{attribute 'linkalways'} 
{attribute 'no_explicit_call' := 'This FB is a CLASS and must be accessed using methods or properties'}
{attribute 'enable_dynamic_creation'}
FUNCTION_BLOCK FINAL NOT_ULINT EXTENDS Node
VAR
	in : _ULINT(0);
	out : _ULINT(0);
END_VAR

METHOD PUBLIC Clone : I_Node
VAR
	pNode : POINTER TO NOT_ULINT;
END_VAR
pNode := __NEW(NOT_ULINT);
Clone := pNode^;
END_METHOD

METHOD FB_init : BOOL
VAR_INPUT
	bInitRetains : BOOL; // if TRUE, the retain variables are initialized (warm start / cold start)
	bInCopyCode : BOOL;  // if TRUE, the instance afterwards gets moved into the copy code (online change)
END_VAR
AddInput('in',THIS^.in);
AddOutput('out', THIS^.out);
END_METHOD

METHOD PROTECTED OnExecute
VAR
END_VAR
out.Value := NOT in.Value;
END_METHOD

END_FUNCTION_BLOCK

(* stored: Version 1.1.0.1, ProductVersion 3.1.4024.15
   POU NOT_ULINT: Id {6a46a913-eabb-4b16-a9d0-e7fe1a2e998c}, SpecialFunc None
   Folder Constructor: Id {a5178578-14a7-4364-9ed2-44a60b2d46d9}
   Method Clone: Id {937ddc2f-052f-4e26-b094-b96bbbc22123}
   Method FB_init: Id {8d2a5437-735e-49f5-bead-c844d7c9e880}
   Method OnExecute: Id {4ce02b46-f51e-40a6-9083-c4b192cc5b10} *)
